FUNCTION_BLOCK AxisControl_MultipleInputSensors
VAR_INPUT
	MethodCall: BOOL;
	EmergencyStopSignal : BOOL;
	Direction : BOOL;
	Sensor_01: BOOL;
	Sensor_02: BOOL;
	TouchSensorRelief: BOOL;
	TOF_Time_MotorControl: TIME;
	TOF_Time_TouchSensorRelief: TIME;
	AutomaticMode: BOOL;
END_VAR

VAR_OUTPUT
	MotorControl_01: BOOL;
	MotorControl_02: BOOL;
	ResetCall: BOOL;
END_VAR

VAR
//FlipFlop
	RS_AxisControl: RS;
	RS_TouchSensorRelief: RS;
//Zeitverzögerung
	TOF_TouchSensorRelief: TOF;
	TOF_MotorControl: TOF;	
//Flanke	
	R_TRIG_MethodCall: R_TRIG;
END_VAR
VAR // added by the converter: edge detectors and wires of the graphical bodies
    _w1 : BOOL;
END_VAR

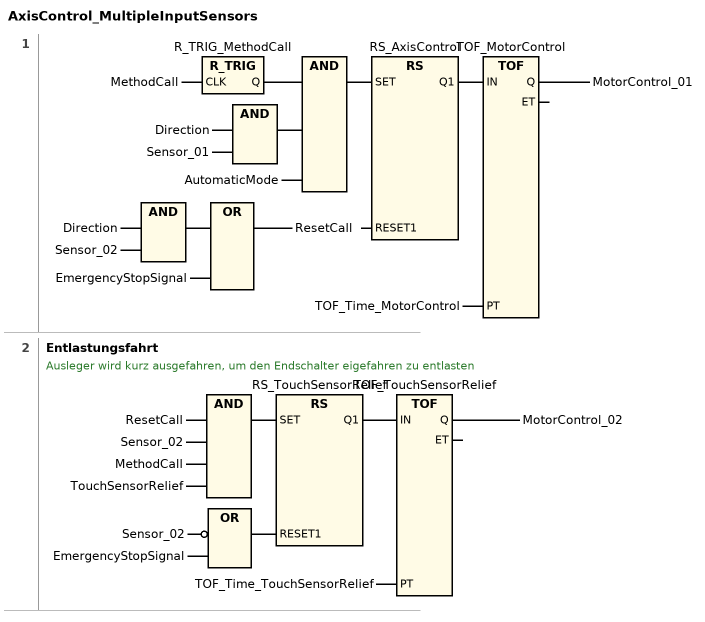
// NETWORK 1
R_TRIG_MethodCall(CLK := MethodCall); // R_TRIG
_w1 := Direction AND Sensor_02 OR EmergencyStopSignal;
ResetCall := _w1;
RS_AxisControl(SET := R_TRIG_MethodCall.Q AND (Direction AND Sensor_01) AND AutomaticMode, RESET1 := _w1); // RS
TOF_MotorControl(IN := RS_AxisControl.Q1, PT := TOF_Time_MotorControl); // TOF
MotorControl_01 := TOF_MotorControl.Q;

// NETWORK 2: Entlastungsfahrt
// Ausleger wird kurz ausgefahren, um den Endschalter eigefahren zu entlasten
RS_TouchSensorRelief(SET := ResetCall AND Sensor_02 AND MethodCall AND TouchSensorRelief, RESET1 := NOT Sensor_02 OR EmergencyStopSignal); // RS
TOF_TouchSensorRelief(IN := RS_TouchSensorRelief.Q1, PT := TOF_Time_TouchSensorRelief); // TOF
MotorControl_02 := TOF_TouchSensorRelief.Q;

END_FUNCTION_BLOCK

(* stored: Version 1.1.0.1, ProductVersion 3.1.4024.15
   POU AxisControl_MultipleInputSensors: Id {7af1c37c-b045-4782-9094-92d73b3f4ccd}, SpecialFunc None *)
